(* PLC project SafeLOGIC-1, BrAutomation SafeDESIGNER  4.3.4.4 *)
(* stored: companyURL http://www.br-automation.com, creationDateTime Wed Jun 16 10:54:11 2021 *)

PROGRAM Main

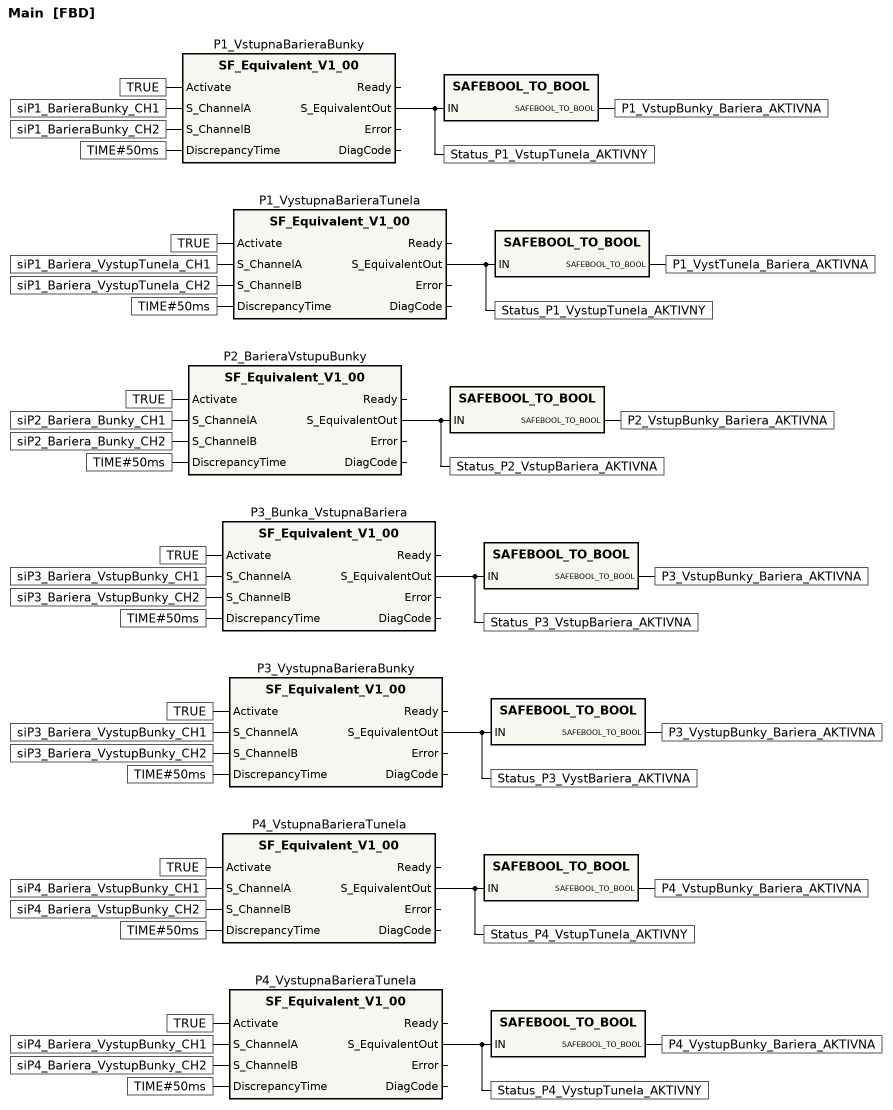
(* FBD diagram, written out as Structured Text *)
P1_VstupnaBarieraBunky(Activate := TRUE, S_ChannelA := siP1_BarieraBunky_CH1, S_ChannelB := siP1_BarieraBunky_CH2, DiscrepancyTime := TIME#50ms);
Status_P1_VstupTunela_AKTIVNY := P1_VstupnaBarieraBunky.S_EquivalentOut;
P1_VstupBunky_Bariera_AKTIVNA := SAFEBOOL_TO_BOOL(P1_VstupnaBarieraBunky.S_EquivalentOut);
P1_VystupnaBarieraTunela(Activate := TRUE, S_ChannelA := siP1_Bariera_VystupTunela_CH1, S_ChannelB := siP1_Bariera_VystupTunela_CH2, DiscrepancyTime := TIME#50ms);
Status_P1_VystupTunela_AKTIVNY := P1_VystupnaBarieraTunela.S_EquivalentOut;
P1_VystTunela_Bariera_AKTIVNA := SAFEBOOL_TO_BOOL(P1_VystupnaBarieraTunela.S_EquivalentOut);
P2_BarieraVstupuBunky(Activate := TRUE, S_ChannelA := siP2_Bariera_Bunky_CH1, S_ChannelB := siP2_Bariera_Bunky_CH2, DiscrepancyTime := TIME#50ms);
Status_P2_VstupBariera_AKTIVNA := P2_BarieraVstupuBunky.S_EquivalentOut;
P2_VstupBunky_Bariera_AKTIVNA := SAFEBOOL_TO_BOOL(P2_BarieraVstupuBunky.S_EquivalentOut);
P3_Bunka_VstupnaBariera(Activate := TRUE, S_ChannelA := siP3_Bariera_VstupBunky_CH1, S_ChannelB := siP3_Bariera_VstupBunky_CH2, DiscrepancyTime := TIME#50ms);
Status_P3_VstupBariera_AKTIVNA := P3_Bunka_VstupnaBariera.S_EquivalentOut;
P3_VstupBunky_Bariera_AKTIVNA := SAFEBOOL_TO_BOOL(P3_Bunka_VstupnaBariera.S_EquivalentOut);
P3_VystupnaBarieraBunky(Activate := TRUE, S_ChannelA := siP3_Bariera_VystupBunky_CH1, S_ChannelB := siP3_Bariera_VystupBunky_CH2, DiscrepancyTime := TIME#50ms);
Status_P3_VystBariera_AKTIVNA := P3_VystupnaBarieraBunky.S_EquivalentOut;
P3_VystupBunky_Bariera_AKTIVNA := SAFEBOOL_TO_BOOL(P3_VystupnaBarieraBunky.S_EquivalentOut);
P4_VstupnaBarieraTunela(Activate := TRUE, S_ChannelA := siP4_Bariera_VstupBunky_CH1, S_ChannelB := siP4_Bariera_VstupBunky_CH2, DiscrepancyTime := TIME#50ms);
Status_P4_VstupTunela_AKTIVNY := P4_VstupnaBarieraTunela.S_EquivalentOut;
P4_VstupBunky_Bariera_AKTIVNA := SAFEBOOL_TO_BOOL(P4_VstupnaBarieraTunela.S_EquivalentOut);
P4_VystupnaBarieraTunela(Activate := TRUE, S_ChannelA := siP4_Bariera_VystupBunky_CH1, S_ChannelB := siP4_Bariera_VystupBunky_CH2, DiscrepancyTime := TIME#50ms);
Status_P4_VystupTunela_AKTIVNY := P4_VystupnaBarieraTunela.S_EquivalentOut;
P4_VystupBunky_Bariera_AKTIVNA := SAFEBOOL_TO_BOOL(P4_VystupnaBarieraTunela.S_EquivalentOut);
END_PROGRAM
